FUNCTION_BLOCK MQTT_SUBSCRIBER_V3
  {SET_ATTRIBUTE(OpcUa, POINT.STARTPOINT)}
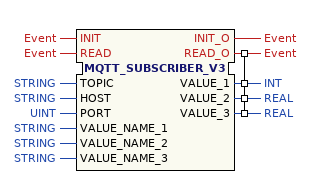
  EVENT_INPUT
    INIT;
    READ;
  END_EVENT
  EVENT_OUTPUT
    INIT_O;
    READ_O WITH VALUE_1, VALUE_2, VALUE_3;
  END_EVENT
  VAR_INPUT
    TOPIC : STRING; {SET_ATTRIBUTE(OpcUa, Constant)}
    HOST : STRING; {SET_ATTRIBUTE(OpcUa, Constant)}
    PORT : UINT; {SET_ATTRIBUTE(OpcUa, Constant)}
    VALUE_NAME_1 : STRING; {SET_ATTRIBUTE(OpcUa, Constant)}
    VALUE_NAME_2 : STRING; {SET_ATTRIBUTE(OpcUa, Constant)}
    VALUE_NAME_3 : STRING; {SET_ATTRIBUTE(OpcUa, Constant)}
  END_VAR
  VAR_OUTPUT
    VALUE_1 : INT; {SET_ATTRIBUTE(OpcUa, Variable)}
    VALUE_2 : REAL; {SET_ATTRIBUTE(OpcUa, Variable)}
    VALUE_3 : REAL; {SET_ATTRIBUTE(OpcUa, Variable)}
  END_VAR
END_FUNCTION_BLOCK
